{attribute 'qualified_only'}
{attribute 'strict'}
{attribute 'to_string'}
TYPE E_STATION_CHECK :
(
	CHECK_NULL,
  STATION_ID_INVALID := 9000,
  REFERENCE_CTRL_INVALID,
  REFERENCE_STATE_INVALID,
  REFERENCE_LIST_ITF_INVALID,
  REFERENCE_MOVER_ITF_INVALID,
  REFERENCE_MOVER_OFFSET_INVALID,
  REFERENCE_PARAMETER_INVALID,
  REFERENCE_MOVER_AXIS_REF_INVALID,

  REFERENCE_MASTER_AXIS_REF_INVALID,
  REFERENCE_GEAR_DATA_INVALID,
  REFERENCE_GEAR_PARAMETER_INVALID,

  CHECK_DONE    := 10_000
);
END_TYPE

(* stored: Version 1.1.0.1
   DUT E_STATION_CHECK: Id {7ddd7694-6e9b-4495-a495-665566aeb33d} *)
